{attribute 'qualified_only'}
VAR_GLOBAL CONSTANT
	// Database ID
	TARGET_DBID : UINT := 1;
END_VAR

(* stored: Version 1.1.0.1, ProductVersion 3.1.4024.12
   GVL GVL: Id {e2f827f0-9ef3-40f7-98dd-013705377226} *)
